// TIA Portal V19 export
VAR_GLOBAL   // PLC tag table "Test"
   bReset AT %I0.0 : Bool;
   bTestFirstScan AT %I0.1 : Bool;
   bTestMonthShift AT %I0.2 : Bool;
   bTEstREset AT %I0.3 : Bool;
END_VAR
VAR_GLOBAL CONSTANT   // user constants
   MAX_DAYS_IN_MONTH : Int := 31;
END_VAR
